FUNCTION_BLOCK C_HTTP_RESPONSE EXTENDS C_HTTP_BASE
VAR_INPUT
END_VAR
VAR_OUTPUT
END_VAR
VAR
	_ResponseCode		: E_HTTP_RESPONSE_CODE;
	_Url				: STRING(255);	
	_c_HttpVersion 		: C_HTTP_VERSION(Major_Version:= 1, Minor_Version:= 1);
	
	_Header 			: ARRAY[0..15] OF C_HTTP_HEADER(Name:= '');
	
	_MessageBody		: T_HTTPSTRING;
END_VAR

PROPERTY Major_Version : uint
GET
Major_Version := _c_HttpVersion.Major;;
END_GET
END_PROPERTY

PROPERTY Minor_Version : uint
GET
Minor_Version := _c_HttpVersion.Minor;
END_GET
END_PROPERTY

END_FUNCTION_BLOCK

(* stored: Version 1.1.0.1, ProductVersion 3.1.4019.2
   POU C_HTTP_RESPONSE: Id {010b61de-28e4-4f7f-b8a2-8dcec89c617c}, SpecialFunc None
   Property Major_Version: Id {afc06728-0a39-4ecb-9385-7a14f5763adb}
   Get Get: Id {c129bdd3-a601-4155-b24a-10f551c1c88c}
   Property Minor_Version: Id {186071c6-7e89-460d-ab59-7a638ff1eb8d}
   Get Get: Id {813ce9fd-3746-4bdc-92f0-55c76cb865ba} *)
